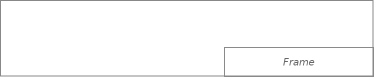
VISUALIZATION Visualization  // 374x77
    Frame (224,47 150x30)
END_VISUALIZATION

(* stored: Version 1.1.0.1
   Visu Visualization: Id {d3ee5358-05ca-4f2a-b6b2-de1c94830cc3} *)
